Fanuc KAREL source: kt00167.KL

-- PROVISIONAL review KL for V1013-1; original PC SHA256 72f33083788a827732a202b27c884c4fa5b91f2198e0aff64cc0bd96d754198a
-- Incomplete behavior may be omitted. Consult companion uncertainty JSON. Do not deploy.
PROGRAM KT00167
%NOLOCKGROUP
VAR
  I1 : INTEGER
  OUT : INTEGER
-- UNRESOLVED_DECL H2 type=002017
BEGIN
  -- UNRESOLVED_PC offsets 5-16; opcodes 2E,23
  -- UNRESOLVED_PC offsets 21-35; opcodes 2E,22,9D,33,B4
  -- UNRESOLVED_PC offsets 40-62; opcodes 21,22,9D,33,B3,56,23
  -- UNRESOLVED_PC offsets 67-71; opcodes 7F
END KT00167
